// Checks if the given generic value is an unsigned integer type.
FUNCTION F_IsUnsignedIntegerGeneric : BOOL // TRUE if the generic value is an unsigned integer type.
VAR_INPUT
	Value : FsCommon.T_Generic; // The generic value to check.
END_VAR

CASE Value.TypeClass OF
	__SYSTEM.TYPE_CLASS.TYPE_BYTE,
	__SYSTEM.TYPE_CLASS.TYPE_WORD,
	__SYSTEM.TYPE_CLASS.TYPE_DWORD,
	__SYSTEM.TYPE_CLASS.TYPE_LWORD,
	__SYSTEM.TYPE_CLASS.TYPE_USINT,
	__SYSTEM.TYPE_CLASS.TYPE_UINT,
	__SYSTEM.TYPE_CLASS.TYPE_UDINT,
	__SYSTEM.TYPE_CLASS.TYPE_ULINT:
		F_IsUnsignedIntegerGeneric := TRUE;
	END_CASE

END_FUNCTION

(* stored: Version 1.1.0.1
   POU F_IsUnsignedIntegerGeneric: Id {aa56935f-0017-0f36-0fe1-2c2990b444f6}, SpecialFunc None *)
